{attribute 'linkalways'} 
{attribute 'no_explicit_call' := 'This FB is a CLASS and must be accessed using methods or properties'}
{attribute 'enable_dynamic_creation'}
FUNCTION_BLOCK Node_F_VN_SetAt_TcVnVector2_UINT EXTENDS VisionNode
VAR
    aElement : _TcVnVector2_UINT;
    ipContainer : _ITcVnContainer;
    nIndex : _ULINT(0);
    hrPrev : _HRESULT(S_OK);
    hresult : _HRESULT(S_OK);
END_VAR

METHOD PUBLIC  Clone : I_Node
VAR
	pNode : POINTER TO Node_F_VN_SetAt_TcVnVector2_UINT;
END_VAR
pNode := __NEW(Node_F_VN_SetAt_TcVnVector2_UINT);
Clone := pNode^;
END_METHOD

METHOD FB_init : BOOL
VAR_INPUT
	bInitRetains : BOOL; // if TRUE, the retain variables are initialized (warm start / cold start)
	bInCopyCode : BOOL;  // if TRUE, the instance afterwards gets moved into the copy code (online change)
END_VAR
AddInput('aElement', aElement);
AddInput('ipContainer', ipContainer);
AddInput('nIndex', nIndex);
AddInput('hrPrev', hrPrev);
AddOutput('ipContainer', ipContainer);
AddOutput('hresult',hresult);
END_METHOD

METHOD PROTECTED OnExecute : HRESULT
hresult.Value := F_VN_SetAt_TcVnVector2_UINT(
    aElement := aElement.Value,
    ipContainer := ipContainer.Value,
    nIndex := nIndex.Value,
    hrPrev:= hrPrev.Value);
END_METHOD

METHOD PUBLIC PreExecutionCheck
VAR_INPUT
	Check : I_PreExecutionChecks;
END_VAR
Check.IsTrue(ipContainer.IsValid, 'ipContainer must be a valid container');
END_METHOD

END_FUNCTION_BLOCK

(* stored: Version 1.1.0.1, ProductVersion 3.1.4024.13
   POU Node_F_VN_SetAt_TcVnVector2_UINT: Id {24501f40-9248-4e8f-a1ef-adfe2ba8cb52}, SpecialFunc None
   Folder Constructor: Id {a978b6d0-8890-46c8-aabb-2ec1edcf20b7}
   Method Clone: Id {eaf772cc-bc82-41f1-8346-f4f9956fcc2e}
   Method FB_init: Id {e46c471b-e944-458c-bf89-b79f89297e64}
   Method OnExecute: Id {4c6495f5-9e3b-4401-9366-1bfecdccca73}
   Method PreExecutionCheck: Id {a372e5b4-21ab-48e7-8480-edf2299d105a} *)
